(* CoDeSys 2.3.9.62 project: Tema2Ejemplo1-Motor.pro *)
(* Libraries: Standard.lib 4.10.05 11:14:46, IecSfc.lib 2.6.14 12:37:46, SYSLIBCALLBACK.LIB*26.9.08 16:43:52 *)

(* POU PLC_PRG, LD *)
PROGRAM PLC_PRG
VAR
	BotonP: BOOL;
	BotonM: BOOL;
	Motor: BOOL;
END_VAR
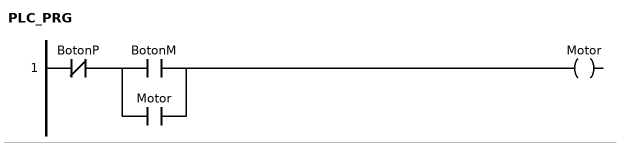
_LD_ (* Ladder Diagram *)
NETWORK 1
	[/BotonP] - { [BotonM] | [Motor] } --- (Motor)
_END_LD_
(* the same logic as Structured Text *)
(* Network 1 *)
Motor := NOT BotonP AND (BotonM OR Motor);
END_PROGRAM

(* Visualisation Botonera
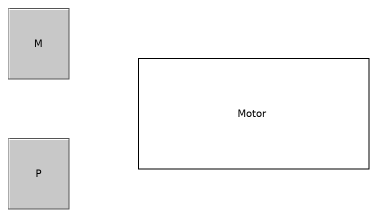
rounded rectangle at (200,80)-(431,191): text "Motor"; shows PLC_PRG.temp1.ET; alarm colour if PLC_PRG.Motor
button at (70,30)-(131,101): text "M"; taps PLC_PRG.BotonM
button at (70,160)-(131,231): text "P"; taps PLC_PRG.BotonP
*)
